// TwinCAT 3 PLC project plc1
// ProgramVersion: 3.1.4024.0
// libraries:
//   Tc2_Standard, * (Beckhoff Automation GmbH)
//   Tc2_System, * (Beckhoff Automation GmbH)
//   Tc3_Mc3PlanarMotion, * (Beckhoff Automation GmbH)
//   Tc3_Module, * (Beckhoff Automation GmbH)
//   Tc3_Physics, * (Beckhoff Automation GmbH)
//   Tc3_XPlanarStandard, * (Beckhoff Automation GmbH)
// project tree:
//   / PlcTask.TcTTO
//   POUs/ MAIN.TcPOU
// real-time tasks:
//   TASK XPlanar Task16: cycle T#250us, priority 1, ADS port 350
//   TASK MC-Task (MET): cycle T#2ms, priority 2, ADS port 351
//   TASK MC-Task (MPT): cycle T#10ms, priority 3, ADS port 352
//   TASK Job Task: cycle default, priority 4
//   TASK PlcTask: cycle T#10ms, priority 20, ADS port 353
// variable links:
//   XPlanar MC Project/Axes/Mover4220_1 <-> TcCOM Objects/XPlanar/Mover4220_1
//     McToIo/STD <-> InputsFromNC3/NC3ToHW
//   TcCOM Objects/XPlanar/Mover4220_1 <-> XPlanar MC Project/Axes/Mover4220_1
//     OutputsToNC3/HWToNC3 <-> IoToMc/STD
//   plc1 Instance <-> XPlanar MC Project/Axes/Mover4220_1
//     PlcTask Inputs/MAIN.Mover01.stMoverRef.MCTOPLC/ACT <-> McToPlc/ACT
//     PlcTask Inputs/MAIN.Mover01.stMoverRef.MCTOPLC/COORDMODE <-> McToPlc/COORDMODE
//     PlcTask Inputs/MAIN.Mover01.stMoverRef.MCTOPLC/SET <-> McToPlc/SET
//     PlcTask Inputs/MAIN.Mover01.stMoverRef.MCTOPLC/SETONTRACK <-> McToPlc/SETONTRACK
//     PlcTask Inputs/MAIN.Mover01.stMoverRef.MCTOPLC/STD <-> McToPlc/STD
//     PlcTask Outputs/MAIN.Mover01.stMoverRef.PLCTOMC/STD <-> PlcToMc/STD
//   plc1 Instance <-> XPlanar MC Project/Groups/Environment
//     PlcTask Inputs/MAIN.XPlanarTable.environment.MCTOPLC_STD <-> McToPlc/STD
//   plc1 Instance <-> XPlanar MC Project/Groups/XPlanar
//     PlcTask Inputs/MAIN.XPlanarTable.group.MCTOPLC_STD <-> McToPlc/STD

CONFIGURATION plc1
    RESOURCE PLC ON TwinCAT3
        TASK PlcTask(INTERVAL := T#10ms, PRIORITY := 20);
        PROGRAM MAIN WITH PlcTask : MAIN;
    END_RESOURCE
END_CONFIGURATION

// ---- POUs/MAIN.TcPOU
PROGRAM MAIN
VAR
	XPlanarTable			: FB_XPlanarSystem;
	Mover01					: FB_XPlanarMoverStandard;
	
	Run						: BOOL;
	xpState					: UDINT;

	xpPos1					: PositionXYC;
	xpPos2					: PositionXYC;

	Pos1x					: LREAL := 120.0;
	Pos1y					: LREAL := 120.0;
	Pos2x					: LREAL := 360.0;
	Pos2y					: LREAL := 120.0;

	fVelocity				: LREAL := 200.0;
	fAcceleration			: LREAL := 1000.0;
	fDeceleration			: LREAL := 1000.0;
	fJerk					: LREAL := 5000.0;
	
END_VAR

CASE xpState OF
0:	// init, wait for Run
	IF Run THEN xpState := xpState + 10; END_IF
		
10:	// enable mover
	Mover01.Enable('Enable at Start');
	xpState := xpState + 10;

20:	// enabled?
	IF Mover01.P_Enable.Done THEN xpState := xpState + 10; END_IF		

30:	// if running set positions
	IF Run THEN
		xpPos1.SetValuesXYC(Pos1x, Pos1y, 0);
		xpPos2.SetValuesXYC(Pos2x, Pos2y, 0);
		xpState := xpState + 10;	
	END_IF
	
40:	// move to pos1
	Mover01.MoveToPosition('Move to Pos1', xpPos1, fVelocity, fAcceleration, fDeceleration, fJerk);
	xpState := xpState + 10;	
	
50:	// at pos1?  continue
	IF Mover01.P_MoveToPosition.Done THEN xpState := xpState + 10; END_IF

60:	// move to pos2
	Mover01.MoveToPosition('Move to Pos2', xpPos2, fVelocity, fAcceleration, fDeceleration, fJerk);
	xpState := xpState + 10;	

70:	// at pos2?  repeat
	IF Mover01.P_MoveToPosition.Done THEN xpState := 30; END_IF
	
END_CASE

Mover01.Cycle();
XPlanarTable.SetMoverStandard(1, Mover01);	
XPlanarTable.Cycle();

END_PROGRAM
